{attribute 'qualified_only'}
VAR_GLOBAL
	Segment	: ARRAY [1..3] OF ST_Segment_Base;
	
	Segment1to3_ShortContactClose	: BOOL;
	Segment1to3_UnShortContactClose	: BOOL;
	LossInterlockPressure			: BOOL;
	PSU1OK							: BOOL;
	
	Fire			: BOOL;
	SegmentCharged	: BOOL;
	TriggerScope	: BOOL;
END_VAR

(* stored: Version 1.1.0.1, ProductVersion 3.1.4024.11
   GVL LCP1_IO: Id {3cac9d65-1e80-419a-9021-db7cad6298e9} *)
